(* Schneider Machine Expert - Basic project Nuevo proyecto, file version 2.7.0.0 *)
(* ProjectInformations: Name=Nuevo proyecto *)

HARDWARE
  Cpu 0: TM221CE24T
  EthernetConfiguration: NetworkName=M221, IpAllocationMode=FixedAddress, IpAddress=0.0.0.0, SubnetMask=0.0.0.0
  SerialLineConfiguration: Baud=Baud19200, Parity=ParityEven, DataBits=DataBits8, StopBits=StopBits1, PhysicalMedium=PhysicalMediumRs485, TransmissionMode=TransmissionModeModbusRtu, SlaveId=1, Addressing=SlaveAddressing
  MastTask: UsePeriodScanMode=false, PeriodScan=100
  FastTask: Period=255
  CpuBehavior: StartingMode=StartAsPreviousState, AutoSaveRamOnEeprom=true, WatchdogPeriod=250

SYMBOLS  (address, symbol, comment, settings)

POU Nuevo POU
  (* SectionNumber=1 *)

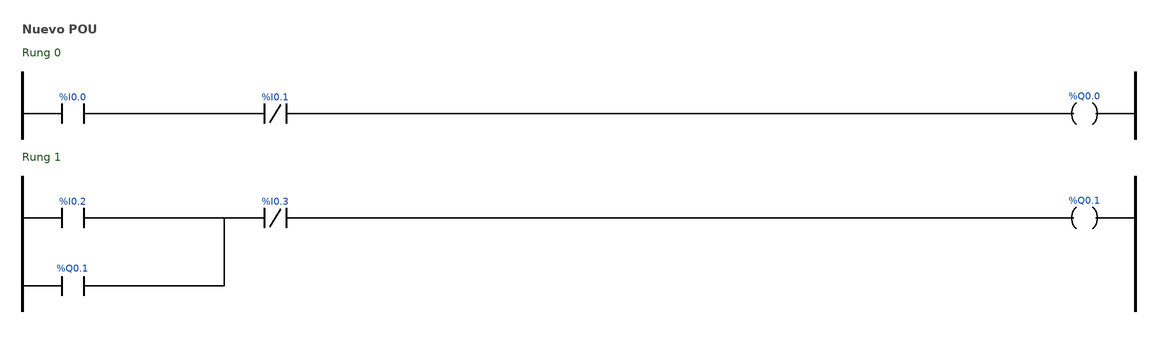

// Rung 0
  LD %I0.0
  ANDN %I0.1
  ST %Q0.0
  // as ST:
  //   %Q0.0 := %I0.0 AND NOT %I0.1;

// Rung 1
  LD %I0.2
  OR %Q0.1
  ANDN %I0.3
  ST %Q0.1
  // as ST:
  //   %Q0.1 := (%I0.2 OR %Q0.1) AND NOT %I0.3;
